(* Logix 5000 project; controller cal1615 1756-L62 rev 20.19; software revision 20.05; part 22 of 81 *)
(* tags used below, declared in another part *)
   FAULT : BOOL;   // Fault AFI
   p01_param_fan_zero_speed : REAL;
   p01_param_open_oven_recirc_sp : REAL;
   p01_param_temp_limit : REAL;   // Machine Parameter Maximum Temperature for Fan Operation
   p01_recipe_active : recipe;   // Active Recipe
   p01r02 : routine;   // System Misc Control
   p01r09_open_oven : BOOL;
   p01r09_pb_global_reset : BOOL;   // System Modes PB: Global Fault Reset
   p02_dint_from_hmi : hmi_dint;
   p11_ai_recirc_rpm : REAL;   // Zone 1 Analog Input Recirc Fan RPM
   p11_ao_recirc_selected_speed : REAL;   // Zone 1 Analog Output Recirc Fan VFD Selected Speed
   p11_di_exh : acs800_di_normal;   // Zone 1 Digital Inputs Exhaust Fan
   p11_di_recirc : acs800_di_normal;   // Zone 1 Digital Inputs Recirc Fan
   p11_di_recirc_fan_mtr_ts : BOOL;   // Zone 1 Digital Input Recirc Fan Motor Thermostat OK
   p11_di_recirc_flow_ok : BOOL;   // Zone 1 Digital Input Recirc Flow OK
   p11_do_recirc : acs800_do_normal;   // Zone 1 Digital Outputs Supply Fan
   p11r01 : routine;   // Zone 1 Main
   p11r02_shutdown_temp : BOOL;   // Zone 1 Misc Control Safe Shutdown Temperature
   p11r20_state : DINT;   // Zone 1 Temperature Control State
   p11r30 : routine;   // Zone 1 Temperature Control
   p11r31 : routine;   // Zone 1 Exhaust VFD
   p11r31_timer_warning : TIMER[5];   // Zone 1 Exhaust VFD Waringing Timer
   p11r32 : routine;   // Zone 1 Recirc VFD
   p11r32_pb_start : BOOL;   // Zone 1 Recirc VFD PB: Start
   p11r32_pb_stop : BOOL;   // Zone 1 Recirc VFD PB: Stop
   p11r32_request_auto_run : BOOL;   // Zone 1 Recirc Fan Run Request
   p11r32_run_permissive : BOOL;   // Zone 1 Recirc VFD Run Permissive
   p11r32_timer_fault : TIMER[5];   // Zone 1 Recirc VFD Fault Timer
   p11r32_timer_warning : TIMER[5];   // Zone 1 Supply VFD Warning Timer
   p11r32_vfd_stopped : BOOL;   // Zone 1 Recirc VFD VFD Stopped
   p12_ai_prs : REAL;   // Zone 2 Analog Input Pressure
   p12_ai_tc01 : REAL;   // Zone 2 Analog Input Control Thermocouple 1
   p12_ai_tc02 : REAL;   // Zone 2 Analog Input Control Thermocouple 2
   p12_dint_to_hmi : DINT[16];   // Zone 2 Temperature Control VFDs On
   p12_param_shutdown_temp : REAL;   // Zone 2 Parameter Zone Shutdown Temperature
   p12_param_zone_pressure : REAL;   // Zone 2 Parameter High Pressure LImit
   p12r01 : routine;   // Zone 2 Main
   p12r02 : routine;   // Zone 2 Misc Control
   p12r02_fault_exists : BOOL;
   p12r02_not_safe_temp : BOOL;   // Zone 2 Misc Control Zone above Safe Temp
   p12r02_safe_temp : BOOL;   // Zone 2 Misc Control Zone Temperature at Safe Temp
   p12r02_shutdown_temp : BOOL;   // Zone 2 Misc Control Safe Shutdown Temperature
   p12r02_timer_fault : TIMER[4];   // Zone 2 Misc Control Fault Delay
   p12r02_timer_safe_temp : TIMER[2];   // Zone 2 Misc Control Chamber SafeTemperature Dwell
   p12r02_timer_warning : TIMER[4];   // Zone 2 Misc Control Warning Delay
   p12r02_unack_fault : BOOL;   // Zone 2 Misc Control Unacknowledged Fault Exists
   p12r02_unack_warning : BOOL;   // Zone 2 Misc Control Unacknowledged Warning Exists
   p12r02_warning_exists : BOOL;
   p12r03 : routine;   // Zone 2 Input
   p12r04 : routine;   // Zone 2 Output
   p12r05 : routine;   // Zone 2 Dint to HMI
   p12r06 : routine;   // Zone 2 Real to HMI
   p12r07 : routine;   // Zone 2 Alarms
   p12r08 : routine;   // Zone 2 Warnings
   p12r09 : routine;   // Zone 2 Modes
   p12r10 : routine;   // Zone 2
   p12r20 : routine;   // Zone 2 Temp Sequence
   p12r30 : routine;   // Zone 2 Temperature Control
   p12r30_pb_zone_off : BOOL;   // Zone 2 Temperature Control PB: Stop Zone Heat Control
   p12r31 : routine;   // Zone 2 Exhaust VFD
   p12r32 : routine;   // Zone 2 Recirc VFD
   p23r02 : routine;   // Impreg Misc Control
(* P11_Zone_1, continued *)

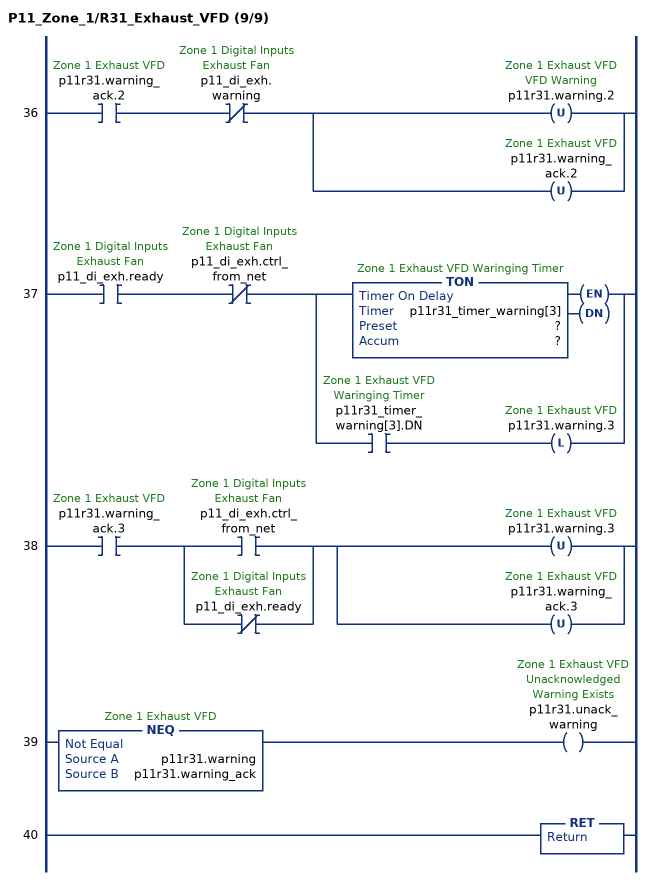
   36: XIC(p11r31.warning_ack.2)XIO(p11_di_exh.warning)[OTU(p11r31.warning.2) ,OTU(p11r31.warning_ack.2) ];
   37: XIC(p11_di_exh.ready)XIO(p11_di_exh.ctrl_from_net)[TON(p11r31_timer_warning[3],?,?) ,XIC(p11r31_timer_warning[3].DN) OTL(p11r31.warning.3) ];
   38: XIC(p11r31.warning_ack.3)[XIC(p11_di_exh.ctrl_from_net) ,XIO(p11_di_exh.ready) ][OTU(p11r31.warning.3) ,OTU(p11r31.warning_ack.3) ];
   39: NEQ(p11r31.warning,p11r31.warning_ack)OTE(p11r31.unack_warning);
   40: RET();
END_ROUTINE

ROUTINE R32_Recirc_VFD   (* ladder *)
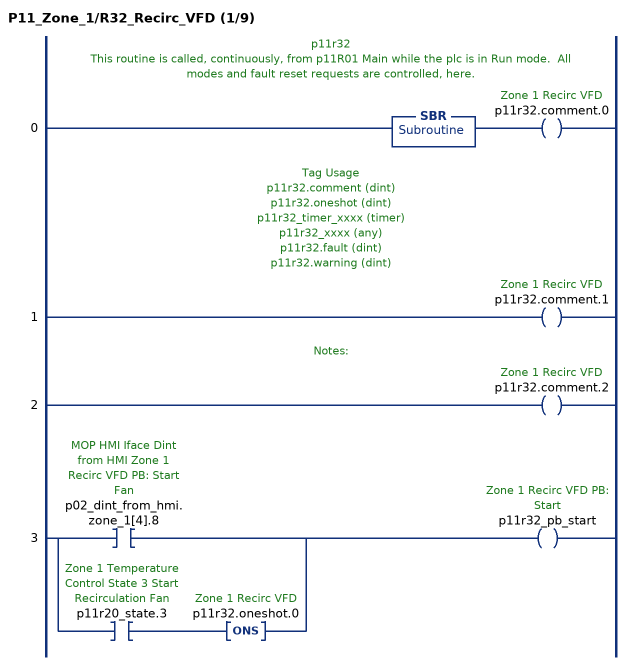
   // p11r32
   // This routine is called, continuously, from p11R01 Main while the plc is in Run mode.  All modes and fault reset requests are controlled, here.
   0: SBR()OTE(p11r32.comment.0);
   // Tag Usage
   // p11r32.comment (dint)
   // p11r32.oneshot (dint)
   // p11r32_timer_xxxx (timer)
   // p11r32_xxxx (any)
   // p11r32.fault (dint)
   // p11r32.warning (dint)
   1: OTE(p11r32.comment.1);
   // Notes:
   2: OTE(p11r32.comment.2);
   3: [XIC(p02_dint_from_hmi.zone_1[4].8) ,XIC(p11r20_state.3) ONS(p11r32.oneshot.0) ]OTE(p11r32_pb_start);
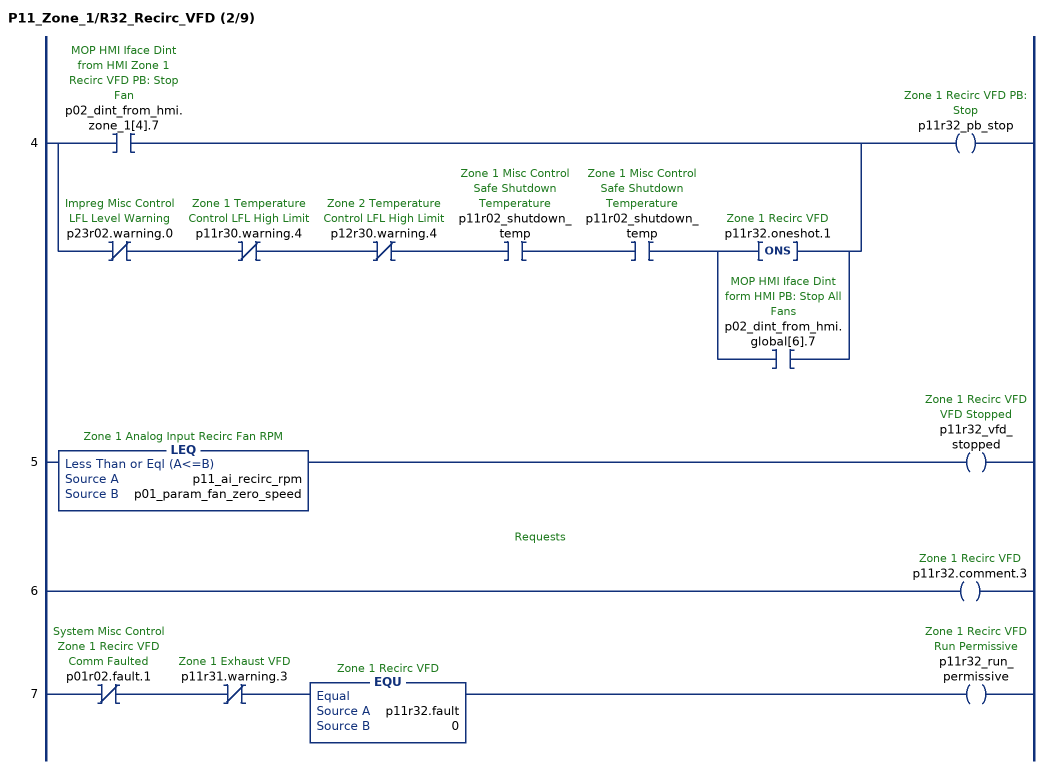
   4: [XIC(p02_dint_from_hmi.zone_1[4].7) ,XIO(p23r02.warning.0) XIO(p11r30.warning.4) XIO(p12r30.warning.4) XIC(p11r02_shutdown_temp) XIC(p11r02_shutdown_temp) [ONS(p11r32.oneshot.1) ,XIC(p02_dint_from_hmi.global[6].7) ] ]OTE(p11r32_pb_stop);
   5: LEQ(p11_ai_recirc_rpm,p01_param_fan_zero_speed)OTE(p11r32_vfd_stopped);
   // Requests
   6: OTE(p11r32.comment.3);
   7: XIO(p01r02.fault.1)XIO(p11r31.warning.3)EQU(p11r32.fault,0)OTE(p11r32_run_permissive);
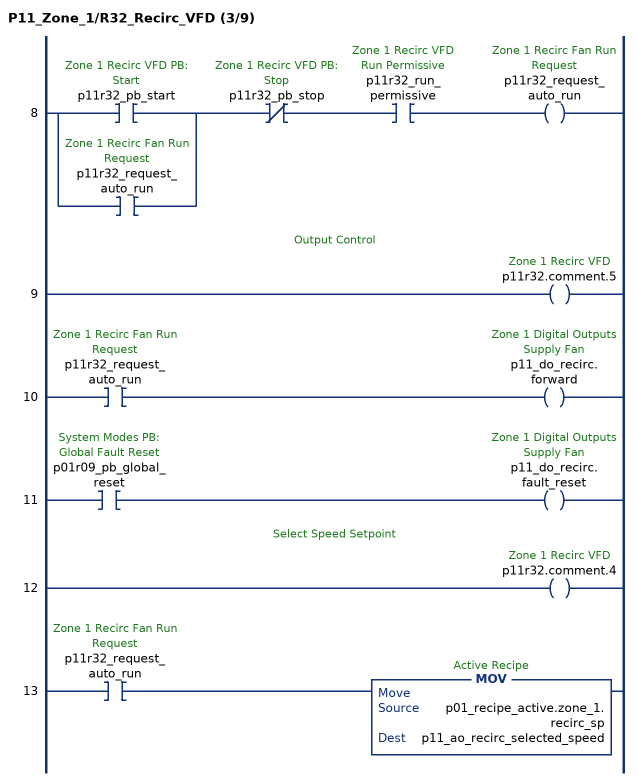
   8: [XIC(p11r32_pb_start) ,XIC(p11r32_request_auto_run) ]XIO(p11r32_pb_stop)XIC(p11r32_run_permissive)OTE(p11r32_request_auto_run);
   // Output Control
   9: OTE(p11r32.comment.5);
   10: XIC(p11r32_request_auto_run)OTE(p11_do_recirc.forward);
   11: XIC(p01r09_pb_global_reset)OTE(p11_do_recirc.fault_reset);
   // Select Speed Setpoint
   12: OTE(p11r32.comment.4);
   13: XIC(p11r32_request_auto_run)MOV(p01_recipe_active.zone_1.recirc_sp,p11_ao_recirc_selected_speed);
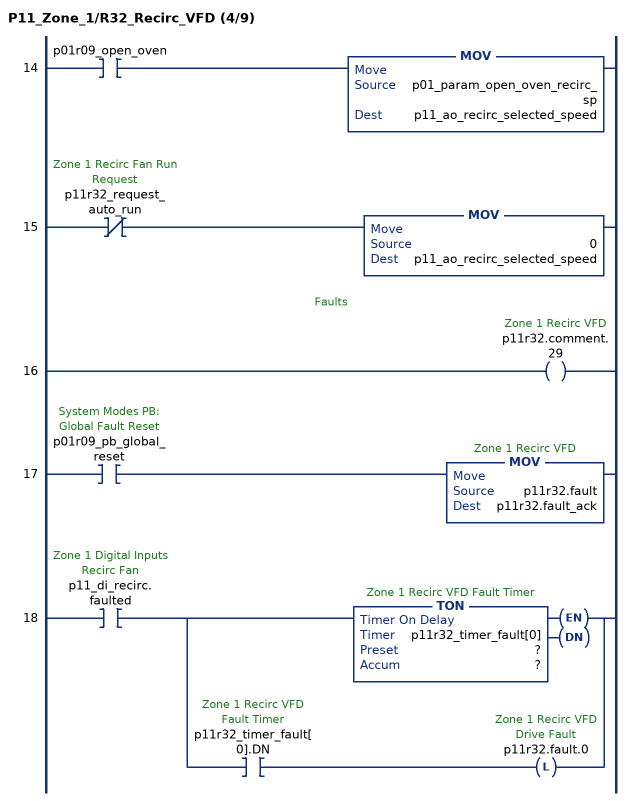
   14: XIC(p01r09_open_oven)MOV(p01_param_open_oven_recirc_sp,p11_ao_recirc_selected_speed);
   15: XIO(p11r32_request_auto_run)MOV(0,p11_ao_recirc_selected_speed);
   // Faults
   16: OTE(p11r32.comment.29);
   17: XIC(p01r09_pb_global_reset)MOV(p11r32.fault,p11r32.fault_ack);
   18: XIC(p11_di_recirc.faulted)[TON(p11r32_timer_fault[0],?,?) ,XIC(p11r32_timer_fault[0].DN) OTL(p11r32.fault.0) ];
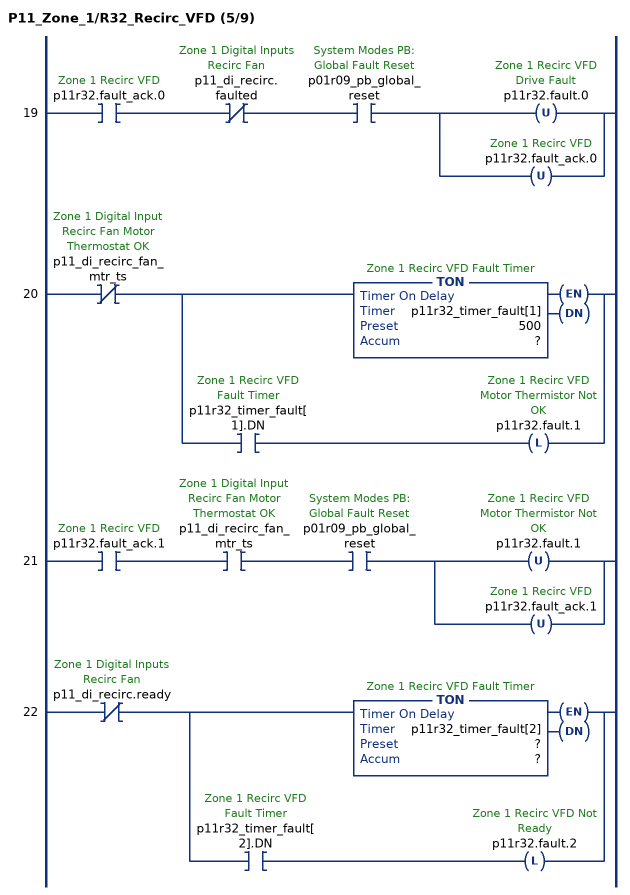
   19: XIC(p11r32.fault_ack.0)XIO(p11_di_recirc.faulted)XIC(p01r09_pb_global_reset)[OTU(p11r32.fault.0) ,OTU(p11r32.fault_ack.0) ];
   20: XIO(p11_di_recirc_fan_mtr_ts)[TON(p11r32_timer_fault[1],?,?) ,XIC(p11r32_timer_fault[1].DN) OTL(p11r32.fault.1) ];
   21: XIC(p11r32.fault_ack.1)XIC(p11_di_recirc_fan_mtr_ts)XIC(p01r09_pb_global_reset)[OTU(p11r32.fault.1) ,OTU(p11r32.fault_ack.1) ];
   22: XIO(p11_di_recirc.ready)[TON(p11r32_timer_fault[2],?,?) ,XIC(p11r32_timer_fault[2].DN) OTL(p11r32.fault.2) ];
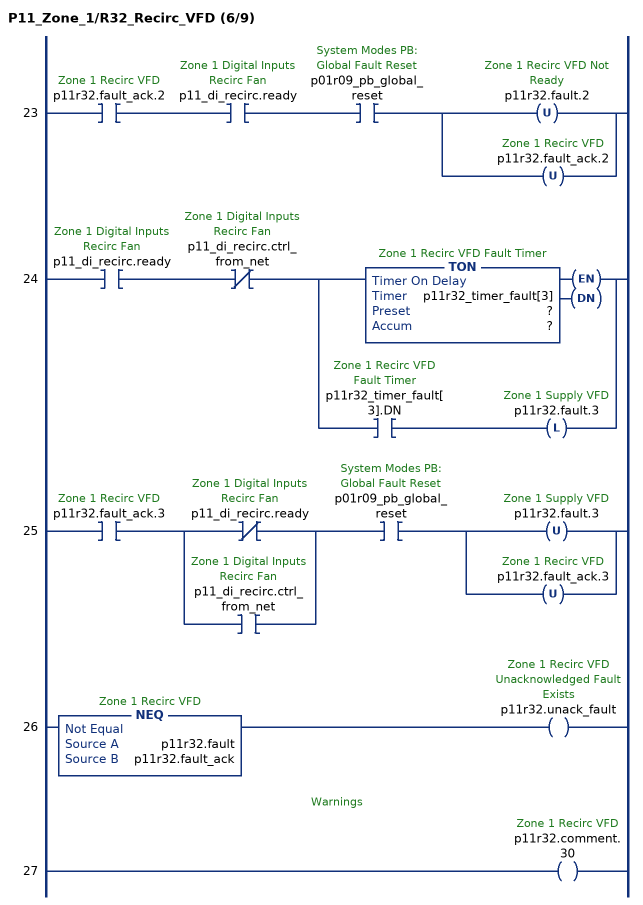
   23: XIC(p11r32.fault_ack.2)XIC(p11_di_recirc.ready)XIC(p01r09_pb_global_reset)[OTU(p11r32.fault.2) ,OTU(p11r32.fault_ack.2) ];
   24: XIC(p11_di_recirc.ready)XIO(p11_di_recirc.ctrl_from_net)[TON(p11r32_timer_fault[3],?,?) ,XIC(p11r32_timer_fault[3].DN) OTL(p11r32.fault.3) ];
   25: XIC(p11r32.fault_ack.3)[XIO(p11_di_recirc.ready) ,XIC(p11_di_recirc.ctrl_from_net) ]XIC(p01r09_pb_global_reset)[OTU(p11r32.fault.3) ,OTU(p11r32.fault_ack.3) ];
   26: NEQ(p11r32.fault,p11r32.fault_ack)OTE(p11r32.unack_fault);
   // Warnings
   27: OTE(p11r32.comment.30);
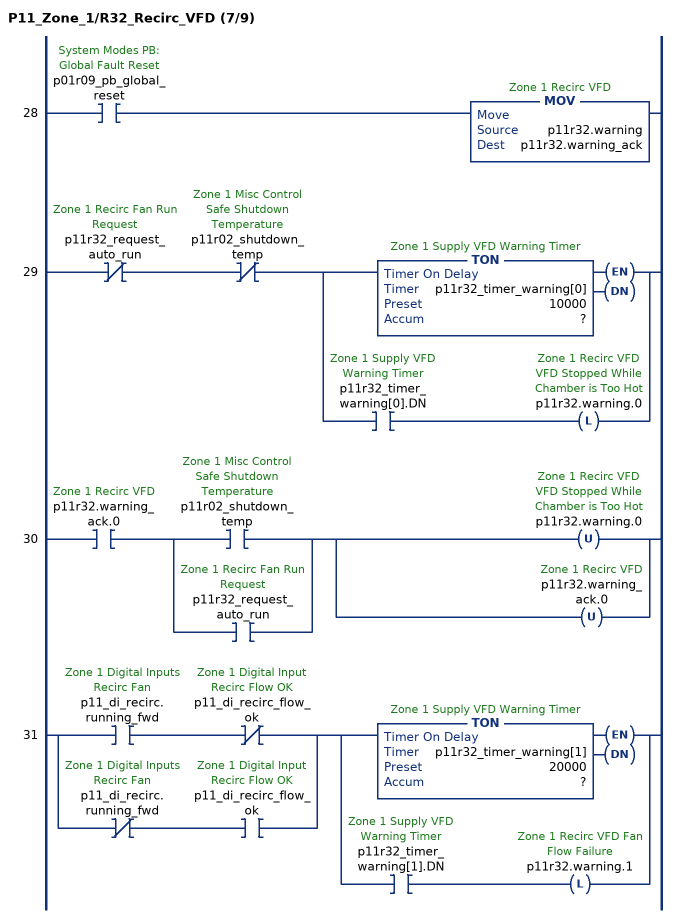
   28: XIC(p01r09_pb_global_reset)MOV(p11r32.warning,p11r32.warning_ack);
   29: XIO(p11r32_request_auto_run)XIO(p11r02_shutdown_temp)[TON(p11r32_timer_warning[0],?,?) ,XIC(p11r32_timer_warning[0].DN) OTL(p11r32.warning.0) ];
   30: XIC(p11r32.warning_ack.0)[XIC(p11r02_shutdown_temp) ,XIC(p11r32_request_auto_run) ][OTU(p11r32.warning.0) ,OTU(p11r32.warning_ack.0) ];
   31: [XIC(p11_di_recirc.running_fwd) XIO(p11_di_recirc_flow_ok) ,XIO(p11_di_recirc.running_fwd) XIC(p11_di_recirc_flow_ok) ][TON(p11r32_timer_warning[1],?,?) ,XIC(p11r32_timer_warning[1].DN) OTL(p11r32.warning.1) ];
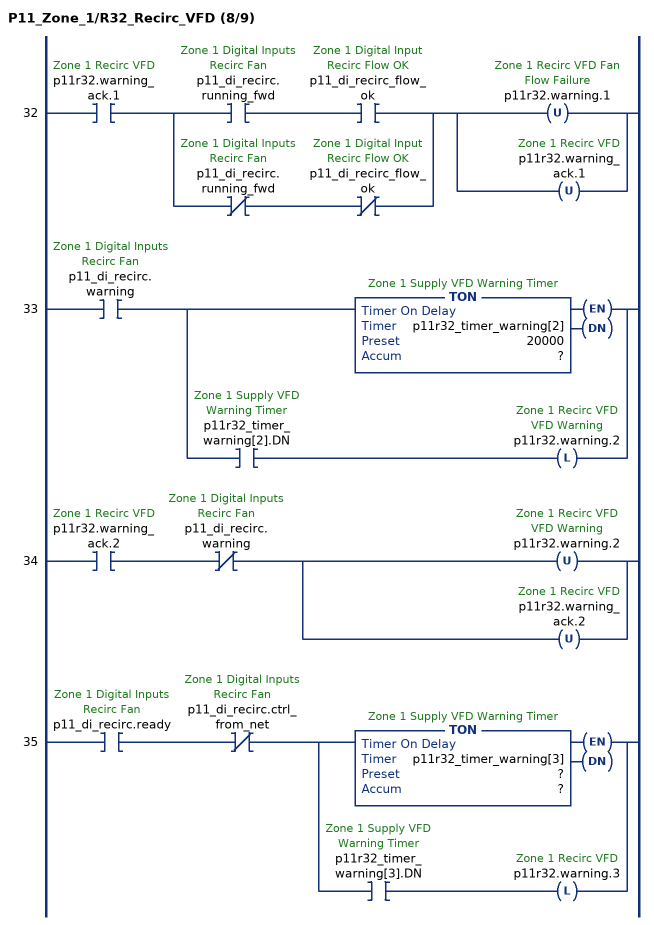
   32: XIC(p11r32.warning_ack.1)[XIC(p11_di_recirc.running_fwd) XIC(p11_di_recirc_flow_ok) ,XIO(p11_di_recirc.running_fwd) XIO(p11_di_recirc_flow_ok) ][OTU(p11r32.warning.1) ,OTU(p11r32.warning_ack.1) ];
   33: XIC(p11_di_recirc.warning)[TON(p11r32_timer_warning[2],?,?) ,XIC(p11r32_timer_warning[2].DN) OTL(p11r32.warning.2) ];
   34: XIC(p11r32.warning_ack.2)XIO(p11_di_recirc.warning)[OTU(p11r32.warning.2) ,OTU(p11r32.warning_ack.2) ];
   35: XIC(p11_di_recirc.ready)XIO(p11_di_recirc.ctrl_from_net)[TON(p11r32_timer_warning[3],?,?) ,XIC(p11r32_timer_warning[3].DN) OTL(p11r32.warning.3) ];
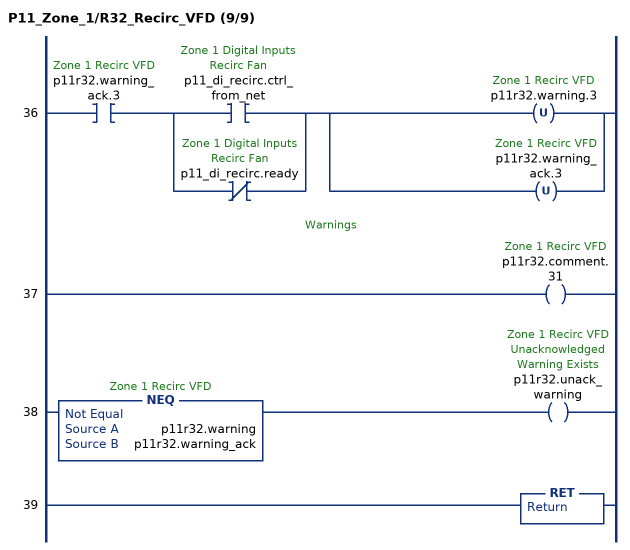
   36: XIC(p11r32.warning_ack.3)[XIC(p11_di_recirc.ctrl_from_net) ,XIO(p11_di_recirc.ready) ][OTU(p11r32.warning.3) ,OTU(p11r32.warning_ack.3) ];
   // Warnings
   37: OTE(p11r32.comment.31);
   38: NEQ(p11r32.warning,p11r32.warning_ack)OTE(p11r32.unack_warning);
   39: RET();
END_ROUTINE
END_PROGRAM

PROGRAM P12_Zone_2   (* main routine R01_Main *)

ROUTINE R01_Main   (* ladder *)
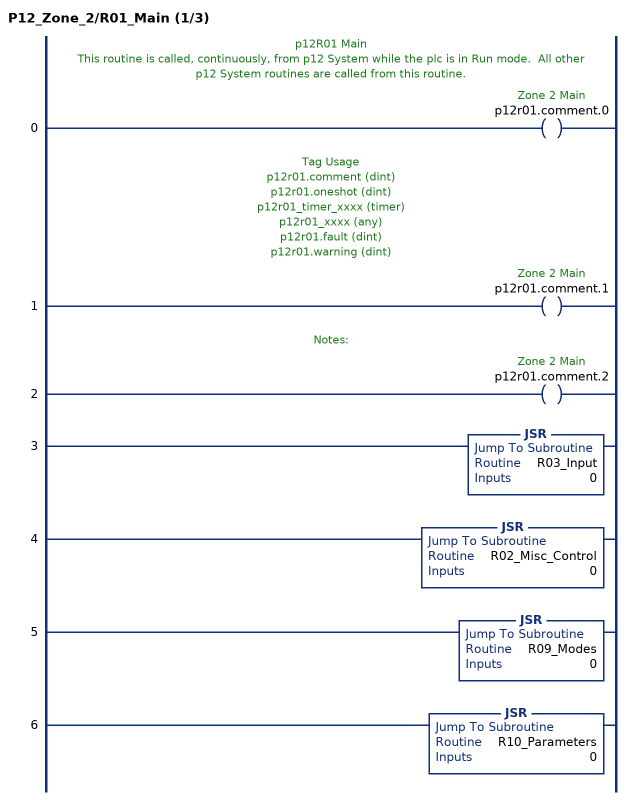
   // p12R01 Main
   // This routine is called, continuously, from p12 System while the plc is in Run mode.  All other p12 System routines are called from this routine.
   0: OTE(p12r01.comment.0);
   // Tag Usage
   // p12r01.comment (dint)
   // p12r01.oneshot (dint)
   // p12r01_timer_xxxx (timer)
   // p12r01_xxxx (any)
   // p12r01.fault (dint)
   // p12r01.warning (dint)
   1: OTE(p12r01.comment.1);
   // Notes:
   2: OTE(p12r01.comment.2);
   3: JSR(R03_Input,0);
   4: JSR(R02_Misc_Control,0);
   5: JSR(R09_Modes,0);
   6: JSR(R10_Parameters,0);
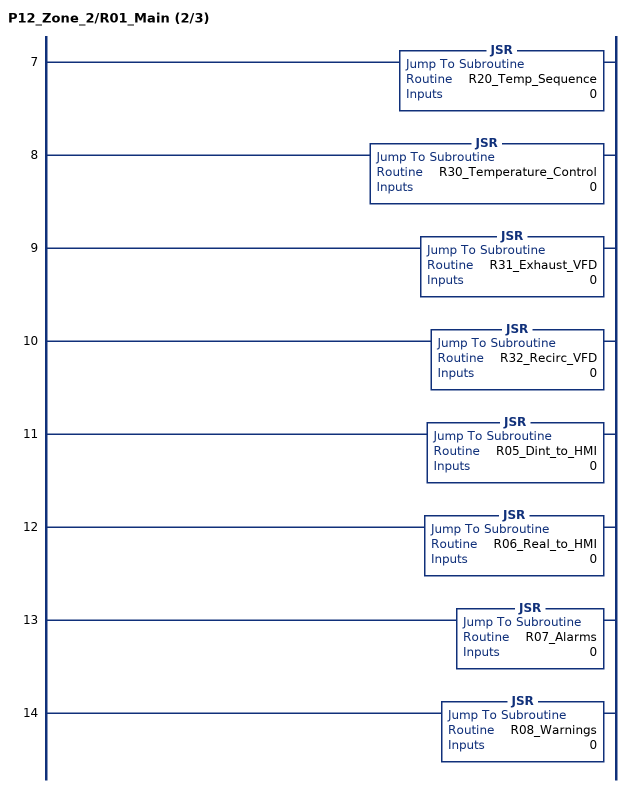
   7: JSR(R20_Temp_Sequence,0);
   8: JSR(R30_Temperature_Control,0);
   9: JSR(R31_Exhaust_VFD,0);
   10: JSR(R32_Recirc_VFD,0);
   11: JSR(R05_Dint_to_HMI,0);
   12: JSR(R06_Real_to_HMI,0);
   13: JSR(R07_Alarms,0);
   14: JSR(R08_Warnings,0);
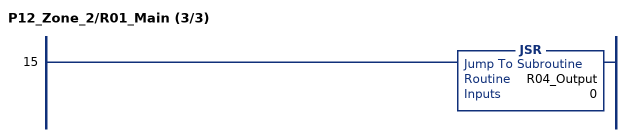
   15: JSR(R04_Output,0);
END_ROUTINE

ROUTINE R02_Misc_Control   (* ladder *)
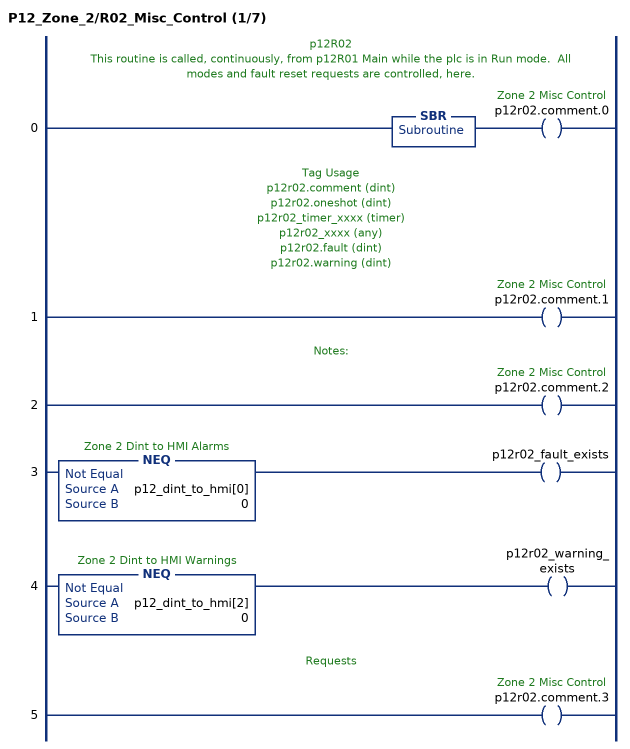
   // p12R02
   // This routine is called, continuously, from p12R01 Main while the plc is in Run mode.  All modes and fault reset requests are controlled, here.
   0: SBR()OTE(p12r02.comment.0);
   // Tag Usage
   // p12r02.comment (dint)
   // p12r02.oneshot (dint)
   // p12r02_timer_xxxx (timer)
   // p12r02_xxxx (any)
   // p12r02.fault (dint)
   // p12r02.warning (dint)
   1: OTE(p12r02.comment.1);
   // Notes:
   2: OTE(p12r02.comment.2);
   3: NEQ(p12_dint_to_hmi[0],0)OTE(p12r02_fault_exists);
   4: NEQ(p12_dint_to_hmi[2],0)OTE(p12r02_warning_exists);
   // Requests
   5: OTE(p12r02.comment.3);
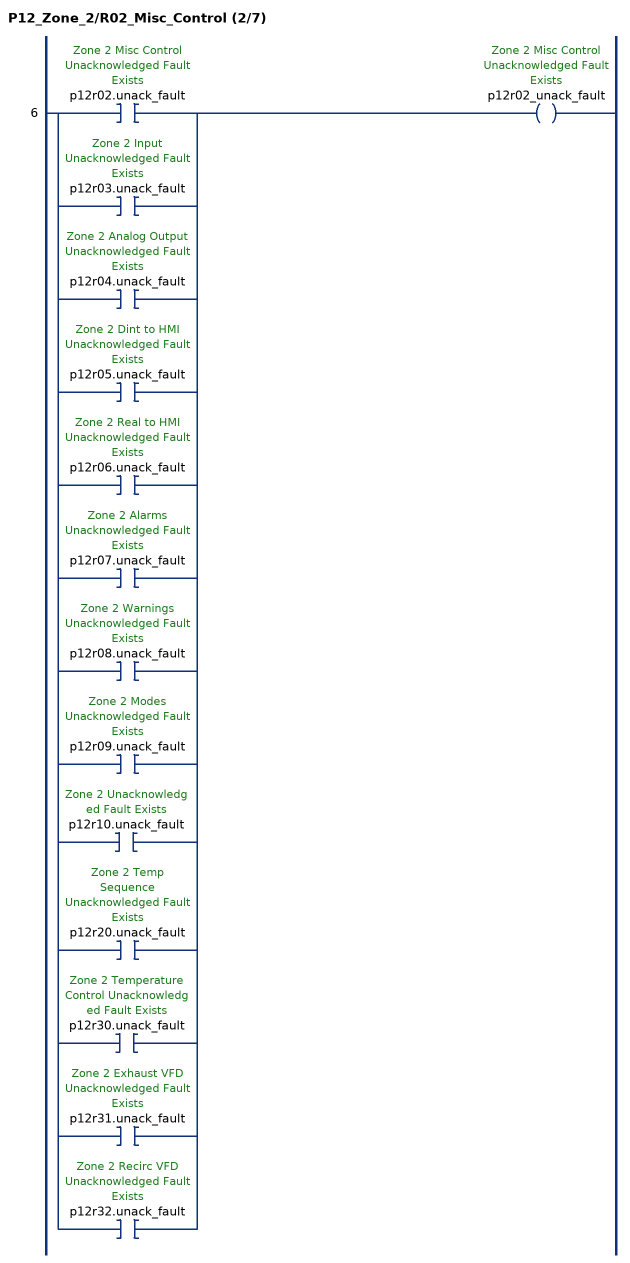
   6: [XIC(p12r02.unack_fault) ,XIC(p12r03.unack_fault) ,XIC(p12r04.unack_fault) ,XIC(p12r05.unack_fault) ,XIC(p12r06.unack_fault) ,XIC(p12r07.unack_fault) ,XIC(p12r08.unack_fault) ,XIC(p12r09.unack_fault) ,XIC(p12r10.unack_fault) ,XIC(p12r20.unack_fault) ,XIC(p12r30.unack_fault) ,XIC(p12r31.unack_fault) ,XIC(p12r32.unack_fault) ]OTE(p12r02_unack_fault);
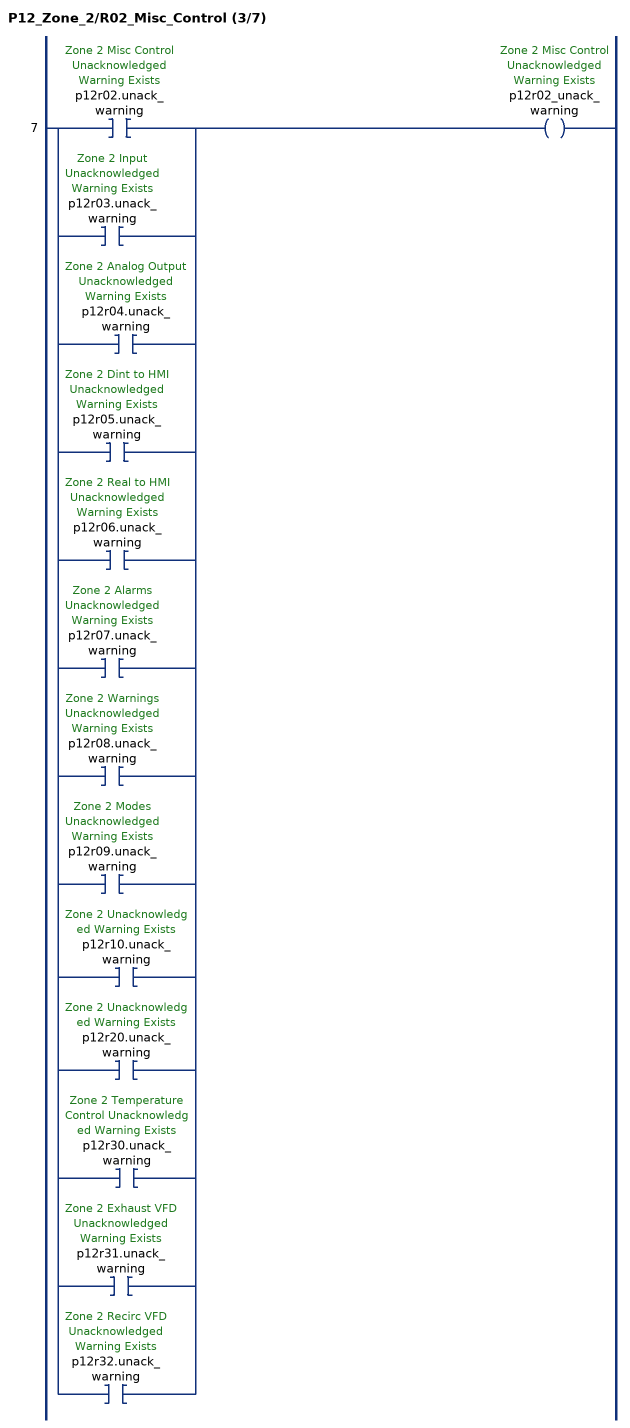
   7: [XIC(p12r02.unack_warning) ,XIC(p12r03.unack_warning) ,XIC(p12r04.unack_warning) ,XIC(p12r05.unack_warning) ,XIC(p12r06.unack_warning) ,XIC(p12r07.unack_warning) ,XIC(p12r08.unack_warning) ,XIC(p12r09.unack_warning) ,XIC(p12r10.unack_warning) ,XIC(p12r20.unack_warning) ,XIC(p12r30.unack_warning) ,XIC(p12r31.unack_warning) ,XIC(p12r32.unack_warning) ]OTE(p12r02_unack_warning);
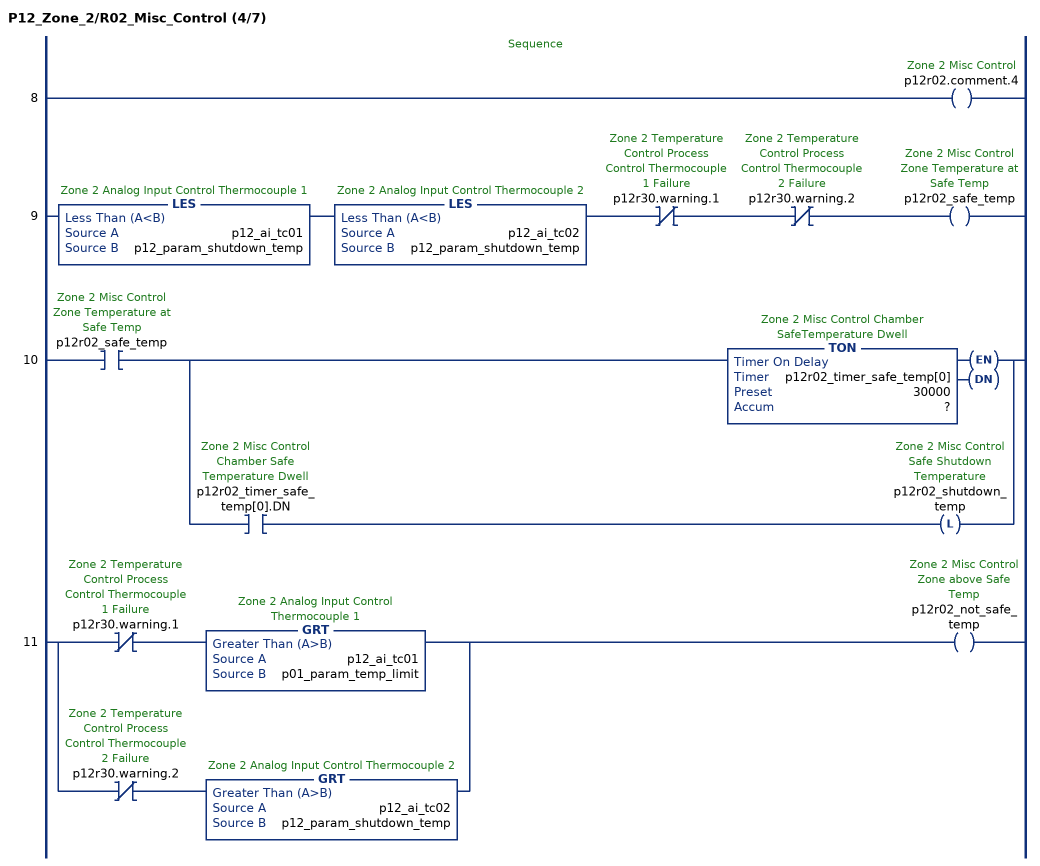
   // Sequence
   8: OTE(p12r02.comment.4);
   9: LES(p12_ai_tc01,p12_param_shutdown_temp)LES(p12_ai_tc02,p12_param_shutdown_temp)XIO(p12r30.warning.1)XIO(p12r30.warning.2)OTE(p12r02_safe_temp);
   10: XIC(p12r02_safe_temp)[TON(p12r02_timer_safe_temp[0],?,?) ,XIC(p12r02_timer_safe_temp[0].DN) OTL(p12r02_shutdown_temp) ];
   11: [XIO(p12r30.warning.1) GRT(p12_ai_tc01,p01_param_temp_limit) ,XIO(p12r30.warning.2) GRT(p12_ai_tc02,p12_param_shutdown_temp) ]OTE(p12r02_not_safe_temp);
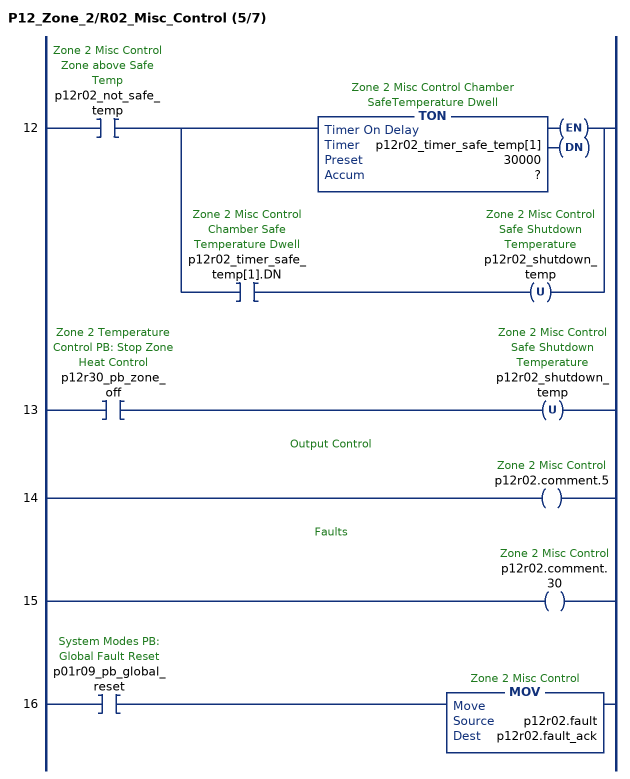
   12: XIC(p12r02_not_safe_temp)[TON(p12r02_timer_safe_temp[1],?,?) ,XIC(p12r02_timer_safe_temp[1].DN) OTU(p12r02_shutdown_temp) ];
   13: XIC(p12r30_pb_zone_off)OTU(p12r02_shutdown_temp);
   // Output Control
   14: OTE(p12r02.comment.5);
   // Faults
   15: OTE(p12r02.comment.30);
   16: XIC(p01r09_pb_global_reset)MOV(p12r02.fault,p12r02.fault_ack);
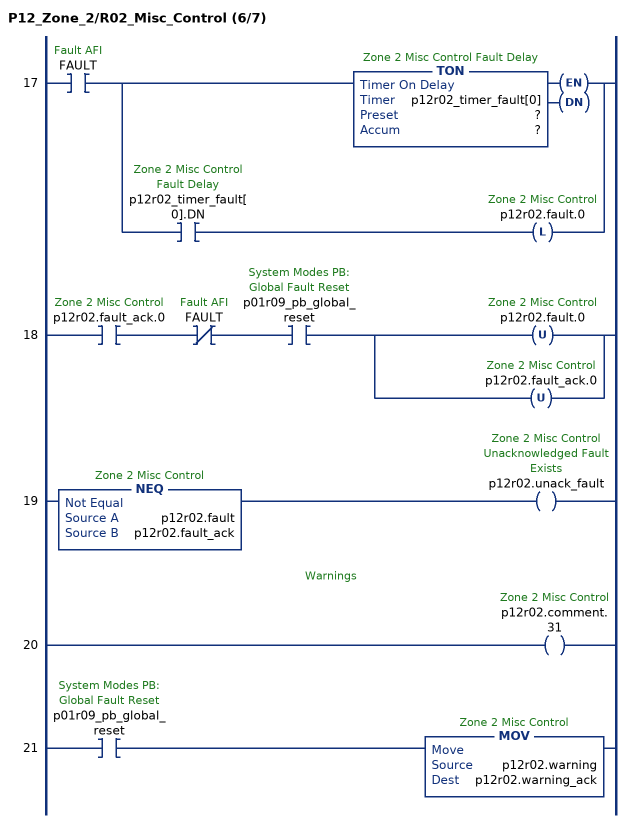
   17: XIC(FAULT)[TON(p12r02_timer_fault[0],?,?) ,XIC(p12r02_timer_fault[0].DN) OTL(p12r02.fault.0) ];
   18: XIC(p12r02.fault_ack.0)XIO(FAULT)XIC(p01r09_pb_global_reset)[OTU(p12r02.fault.0) ,OTU(p12r02.fault_ack.0) ];
   19: NEQ(p12r02.fault,p12r02.fault_ack)OTE(p12r02.unack_fault);
   // Warnings
   20: OTE(p12r02.comment.31);
   21: XIC(p01r09_pb_global_reset)MOV(p12r02.warning,p12r02.warning_ack);
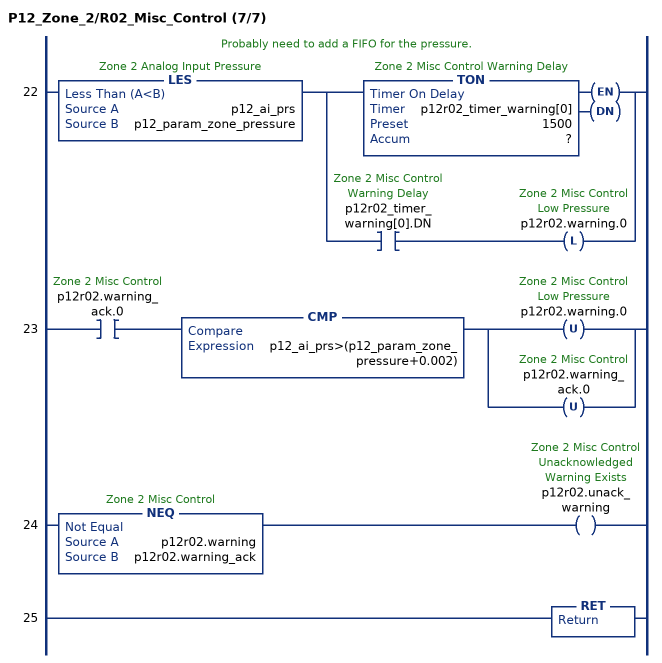
   // Probably need to add a FIFO for the pressure.
   22: LES(p12_ai_prs,p12_param_zone_pressure)[TON(p12r02_timer_warning[0],?,?) ,XIC(p12r02_timer_warning[0].DN) OTL(p12r02.warning.0) ];
   23: XIC(p12r02.warning_ack.0)CMP(p12_ai_prs>(p12_param_zone_pressure+0.002))[OTU(p12r02.warning.0) ,OTU(p12r02.warning_ack.0) ];
   24: NEQ(p12r02.warning,p12r02.warning_ack)OTE(p12r02.unack_warning);
   25: RET();
END_ROUTINE
